(* IEC 61131-3 sources: FDTools/src/Ar/FDTools, 7 files *)

(* ---- DeviceLinker.typ ---- *)
(*
* File: DeviceLinker.typ
* Copyright (c) 2023 Loupe
* https://loupe.team
*
* This file is part of FDTools, licensed under the MIT License.
*
*)

TYPE
	USB_typ : 	STRUCT
		IN : USB_IN_typ;
		OUT : USB_OUT_typ;
		Internal : USB_Internal_typ;
	END_STRUCT;
	USB_IN_typ : 	STRUCT
		PAR : USB_PAR_typ;
		CMD : USB_CMD_typ;
	END_STRUCT;
	USB_PAR_typ : 	STRUCT
		filterInterfaceClass : UINT;
		filterInterfaceSubClass : UINT;
	END_STRUCT;
	USB_CMD_typ : 	STRUCT
		Refresh : BOOL;
		AcknowledgeError : BOOL;
	END_STRUCT;
	USB_OUT_typ : 	STRUCT
		STAT : USB_STAT_typ;
		Interface : ARRAY[0..USB_MAI_NODES]OF STRING[80];
		NumInterfaces : USINT;
		MassStorageDevice : ARRAY[0..USB_MAI_NODES]OF STRING[80];
		NumMassStorages : USINT;
	END_STRUCT;
	USB_STAT_typ : 	STRUCT
		Done : BOOL;
		Busy : BOOL;
		Error : BOOL;
		ErrorID : UINT;
		ErrorString : STRING[80];
	END_STRUCT;
	USB_Internal_typ : 	STRUCT
		State : USB_STATE;
		CMD : USB_CMD_typ;
		STAT : USB_STAT_typ;
		NodeIDList : ARRAY[0..USB_MAI_NODES]OF UDINT;
		NodeList : ARRAY[0..USB_MAI_NODES]OF usbNode_typ;
		DescriptorList : ARRAY[0..USB_MAI_NODES]OF usbDeviceDescr_typ;
		FUB : USB_Internal_FUB_typ;
		NodeIndex : INT;
		AuxInterfaces : ARRAY[0..USB_MAI_NODES]OF STRING[80];
		NumAuxInterface : USINT;
		MassStorageDevices : ARRAY[0..USB_MAI_NODES]OF STRING[80];
		NumMassStorage : USINT;
		RefreshTimer : TON;
	END_STRUCT;
	USB_Internal_FUB_typ : 	STRUCT
		NodeListGet : UsbNodeListGet;
		NodeGet : UsbNodeGet;
		DescriptorGet : UsbDescriptorGet;
	END_STRUCT;
	USB_Selector_Internal_typ : 	STRUCT
		DeviceString : STRING[80];
		iSelectedDevice : STRING[LIST_BOX_STRING_SIZE];
		FileDeviceManager : FileDeviceMgr;
		USBIndex : DINT;
		USBIndexString : STRING[80];
	END_STRUCT;
	FileDeviceMgr_Internal_typ : 	STRUCT
		DevLinkFub : DevLink;
		DevUnlinkFub : DevUnlink;
		iExecute : BOOL;
	END_STRUCT;
	USB_STATE :
		(
		USB_ST_IDLE,
		USB_ST_NODES_GET,
		USB_ST_NODES_READ,
		USB_ST_DESCRIPTORS_READ,
		USB_ST_ERROR,
		USB_ST_
		);
END_TYPE

(* ---- Types.typ ---- *)
(*
* File: Types.typ
* Copyright (c) 2023 Loupe
* https://loupe.team
*
* This file is part of FDTools, licensed under the MIT License.
*
*)

TYPE

END_TYPE

(* ---- USBList.st ---- *)
(*
* File: USBList.st
* Copyright (c) 2023 Loupe
* https://loupe.team
*
* This file is part of FDTools, licensed under the MIT License.
*
*)

(* List all USB nodes *)
FUNCTION USBList

	IF NOT USB.IN.CMD.Refresh AND USB.Internal.CMD.Refresh OR USB.IN.CMD.AcknowledgeError THEN

		USB.IN.CMD.AcknowledgeError:=	0;

		USB.Internal.CMD.Refresh:=0;

		//Reset status
		USB.Internal.STAT.Done:=		0;
		USB.Internal.STAT.Error:=		0;
		USB.Internal.STAT.ErrorID:=		0;
		USB.Internal.STAT.ErrorString:=	'';

	END_IF

	CASE USB.Internal.State OF

		USB_ST_IDLE:

			USB.Internal.STAT.Busy:=		0;

			IF USB.IN.CMD.Refresh AND NOT USB.Internal.CMD.Refresh THEN

				USB.Internal.CMD.Refresh:= 1;

				USB.Internal.State:=	USB_ST_NODES_GET;

				//Reset statuses
				USB.Internal.STAT.Busy:=	1;
				USB.Internal.STAT.Done:=	0;

				//Reset outputs
				USB.Internal.NumMassStorage:=	0;
				USB.Internal.NumAuxInterface:=	0;
				brsmemset(ADR(USB.Internal.MassStorageDevices),0,SIZEOF(USB.Internal.MassStorageDevices));
				brsmemset(ADR(USB.Internal.AuxInterfaces),0,SIZEOF(USB.Internal.AuxInterfaces));

				//Clear out old node data
				brsmemset(ADR(USB.Internal.NodeList),0,SIZEOF(USB.Internal.NodeList));
				brsmemset(ADR(USB.Internal.DescriptorList),0,SIZEOF(USB.Internal.DescriptorList));

			END_IF

		USB_ST_NODES_GET:

			USB.Internal.FUB.NodeListGet.enable:=					1;

			CASE USB.Internal.FUB.NodeListGet.status OF

				ERR_OK:

					USB.Internal.State:=	USB_ST_NODES_READ;

				asusbERR_USB_NOTFOUND:

					USB.Internal.State:=	USB_ST_IDLE;
					USB.Internal.STAT.Done:=	1;

					brsmemcpy(ADR(USB.OUT.Interface),ADR(USB.Internal.AuxInterfaces),SIZEOF(USB.OUT.Interface));
					brsmemcpy(ADR(USB.OUT.MassStorageDevice),ADR(USB.Internal.MassStorageDevices),SIZEOF(USB.OUT.MassStorageDevice));

				ERR_FUB_ENABLE_FALSE,
				ERR_FUB_BUSY:

				ELSE

					USB.Internal.STAT.Error:=		1;
					USB.Internal.STAT.ErrorID:=		USB.Internal.FUB.NodeListGet.status;
					USB.Internal.STAT.ErrorString:=	'Error getting node list';
					USB.Internal.State:=			USB_ST_ERROR;

			END_CASE

		USB_ST_NODES_READ:

			CASE USB.Internal.FUB.NodeGet.status OF

				ERR_OK:

					IF USB.Internal.NodeList[USB.Internal.NodeIndex].interfaceClass = 8 THEN
						USB.Internal.MassStorageDevices[USB.Internal.NumMassStorage]:=	USB.Internal.NodeList[USB.Internal.NodeIndex].ifName;
						USB.Internal.NumMassStorage:=	USB.Internal.NumMassStorage+1;
					ELSIF USB.Internal.NodeList[USB.Internal.NodeIndex].interfaceClass = 255 THEN
						USB.Internal.AuxInterfaces[USB.Internal.NumAuxInterface]:=	USB.Internal.NodeList[USB.Internal.NodeIndex].ifName;
						USB.Internal.NumAuxInterface:=	USB.Internal.NumAuxInterface+1;
					END_IF

					USB.Internal.NodeIndex:=USB.Internal.NodeIndex+1;

					IF USB.Internal.FUB.NodeListGet.listNodes > 0
						AND USB.Internal.FUB.NodeListGet.listNodes > USB.Internal.NodeIndex
						AND USB.Internal.NodeIndex < SIZEOF(USB.Internal.NodeIDList)/SIZEOF(USB.Internal.NodeIDList[0]) THEN

						USB.Internal.FUB.NodeGet.enable:=		1;

					ELSE

						USB.Internal.State:=	USB_ST_DESCRIPTORS_READ;

					END_IF

				ERR_FUB_BUSY:

					//WAIT
					USB.Internal.FUB.NodeGet.enable:=		1;

				ERR_FUB_ENABLE_FALSE:

					USB.Internal.NodeIndex:= 0;
					USB.Internal.FUB.NodeGet.enable:=		1;

				ELSE

					USB.Internal.STAT.Error:=		1;
					USB.Internal.STAT.ErrorID:=		USB.Internal.FUB.NodeGet.status;
					USB.Internal.STAT.ErrorString:=	'Error reading nodes';
					USB.Internal.State:=			USB_ST_ERROR;

			END_CASE

		USB_ST_DESCRIPTORS_READ:

			CASE USB.Internal.FUB.DescriptorGet.status OF
				ERR_OK:

					USB.Internal.NodeIndex:=USB.Internal.NodeIndex+1;

					IF USB.Internal.FUB.NodeListGet.listNodes > 0
						AND USB.Internal.FUB.NodeListGet.listNodes > USB.Internal.NodeIndex
						AND USB.Internal.NodeIndex < SIZEOF(USB.Internal.NodeIDList)/SIZEOF(USB.Internal.NodeIDList[0]) THEN

						USB.Internal.FUB.DescriptorGet.enable:=		1;

					ELSE

						USB.Internal.State:=		USB_ST_IDLE;
						USB.Internal.STAT.Done:=	1;

						brsmemcpy(ADR(USB.OUT.Interface),ADR(USB.Internal.AuxInterfaces),SIZEOF(USB.OUT.Interface));
						brsmemcpy(ADR(USB.OUT.MassStorageDevice),ADR(USB.Internal.MassStorageDevices),SIZEOF(USB.OUT.MassStorageDevice));

						USB.OUT.NumInterfaces:= USB.Internal.NumAuxInterface;
						USB.OUT.NumMassStorages:= USB.Internal.NumMassStorage;

					END_IF

				ERR_FUB_BUSY:

					//WAIT
					USB.Internal.FUB.DescriptorGet.enable:=		1;

				ERR_FUB_ENABLE_FALSE:

					USB.Internal.NodeIndex:= 0;
					USB.Internal.FUB.DescriptorGet.enable:=		1;

				ELSE

					USB.Internal.STAT.Error:=		1;
					USB.Internal.STAT.ErrorID:=		USB.Internal.FUB.DescriptorGet.status;
					USB.Internal.STAT.ErrorString:=	'Error reading node descriptions';
					USB.Internal.State:=			USB_ST_ERROR;

			END_CASE

		USB_ST_ERROR:

			USB.Internal.State:=			USB_ST_IDLE;

	END_CASE

	USB.Internal.RefreshTimer.IN:=	USB.Internal.STAT.Done;
	USB.Internal.RefreshTimer.PT:=	T#3s;
	USB.Internal.RefreshTimer();
	IF USB.Internal.RefreshTimer.Q THEN
		USB.Internal.CMD.Refresh:=	0;
	END_IF

	USB.Internal.FUB.NodeListGet.pBuffer:= 					ADR(USB.Internal.NodeIDList[0]);
	USB.Internal.FUB.NodeListGet.bufferSize:= 				SIZEOF(USB.Internal.NodeIDList);
	USB.Internal.FUB.NodeListGet.filterInterfaceClass:= 	USB.IN.PAR.filterInterfaceClass;
	USB.Internal.FUB.NodeListGet.filterInterfaceSubClass:= 	USB.IN.PAR.filterInterfaceSubClass;
	USB.Internal.FUB.NodeListGet();
	USB.Internal.FUB.NodeListGet.enable:=	0;

	USB.Internal.FUB.NodeGet.nodeId:= 		USB.Internal.NodeIDList[USB.Internal.NodeIndex];
	USB.Internal.FUB.NodeGet.pBuffer:= 		ADR(USB.Internal.NodeList[USB.Internal.NodeIndex]);
	USB.Internal.FUB.NodeGet.bufferSize:= 	SIZEOF(USB.Internal.NodeList[0]);
	USB.Internal.FUB.NodeGet();
	USB.Internal.FUB.NodeGet.enable:=	0;

	USB.Internal.FUB.DescriptorGet.nodeId:= 		USB.Internal.NodeIDList[USB.Internal.NodeIndex];
	USB.Internal.FUB.DescriptorGet.pBuffer:= 		ADR(USB.Internal.DescriptorList[USB.Internal.NodeIndex]);
	USB.Internal.FUB.DescriptorGet.bufferSize:= 	SIZEOF(USB.Internal.DescriptorList[0]);
	//	USB.Internal.FUB.DescriptorGet.descriptorIndex
	//	USB.Internal.FUB.DescriptorGet.descriptorType
	//	USB.Internal.FUB.DescriptorGet.languageId
	//	USB.Internal.FUB.DescriptorGet.requestType
	USB.Internal.FUB.DescriptorGet.descriptorType:= 2;
	USB.Internal.FUB.DescriptorGet();
	USB.Internal.FUB.DescriptorGet.enable:=	0;

	USB.OUT.STAT:=	USB.Internal.STAT;

	USBList:=	USB.OUT.STAT.Done;

END_FUNCTION

(* ---- FDTools.fun ---- *)
(*
* File: FDTools.fun
* Copyright (c) 2023 Loupe
* https://loupe.team
*
* This file is part of FDTools, licensed under the MIT License.
*
*)

FUNCTION USBList : BOOL (*List all USB nodes*) (*$GROUP=User,$GROUPICON=usbms01.front.png*)
	VAR_INPUT
		USB : USB_typ;
	END_VAR
END_FUNCTION

FUNCTION_BLOCK FileDeviceSelector (*Allows the user to select between multiple sources for a file device*) (*$GROUP=User*)
	VAR_INPUT
		Enable : BOOL; (*Enable this function block*)
		FileDevice : STRING[80]; (*File device to link the selected hardware to*)
		pConfiguredDevice : UDINT; (*OPTIONAL: Connect to remnant string variable to reconnect on startup*)
		pUSBList : REFERENCE TO USB_typ; (*OPTIONAL: ADR to USB_typ to populate the list with USB devices*)
		pDirectory : REFERENCE TO STRING[80]; (*OPTIONAL: ADR of String containing the directory to connect to on the CF card*)
		pNetworkConfiguration : REFERENCE TO STRING[80]; (*OPTIONAL: ADR of String containing the network configuration to connect to*)
		Selector : ListBoxFub; (*HMI Connections. Connect this structure to HMI elements to display the results and allow users to select devices.*)
	END_VAR
	VAR_OUTPUT
		Locations : ARRAY[0..12] OF STRING[LIST_BOX_STRING_SIZE]; (*HMI Connections. Connect this array to Listbox or Dropdown to display the results and allow the user to select a device.*)
		status : UINT; (*Status of internal functions*)
		handle : UDINT; (*Handle to unlink in exit routine*)
	END_VAR
	VAR
		internal : USB_Selector_Internal_typ;
		TempString : REFERENCE TO STRING[80];
	END_VAR
END_FUNCTION_BLOCK

FUNCTION_BLOCK FileDeviceMgr (*Links/Unlinks file devices*) (*$GROUP=User*)
	VAR_INPUT
		Execute : BOOL; (*Execute a DevLink*)
		pDevice : UDINT; (*File device to link to hardware*)
		pParam : UDINT; (*Parameter string. See Devlink Help.*)
	END_VAR
	VAR_OUTPUT
		busy : BOOL; (*The function block is working*)
		done : BOOL; (*The function block completed successfully*)
		error : BOOL; (*Error has occured*)
		status : UINT; (*status of devlink/unlink*)
		handle : UDINT; (*Handle to unlink in exit routine*)
	END_VAR
	VAR
		internal : FileDeviceMgr_Internal_typ;
	END_VAR
END_FUNCTION_BLOCK

(* ---- FileDeviceMgr.st ---- *)
(*
* File: FileDeviceMgr.st
* Copyright (c) 2023 Loupe
* https://loupe.team
*
* This file is part of FDTools, licensed under the MIT License.
*
*)

(* Links/Unlinks file devices *)
FUNCTION_BLOCK FileDeviceMgr

	//If execute is false, reset all statuses
	IF NOT Execute THEN

		busy:= 		0;
		done:= 		0;
		status:=	0;
		error:=		0;
		internal.iExecute:=	0;

	END_IF

	//If we have a handle it means that we have devlinked
	//Completion means the user has made a change
	//If so, unlink, then link to the new one
	IF internal.DevUnlinkFub.handle <> 0 AND NOT internal.iExecute AND Execute THEN

		busy:= 		1;
		done:= 		0;
		error:=		0;
		status:= ERR_FUB_BUSY;

		internal.iExecute:=	1;
		internal.DevUnlinkFub.enable:=	1;

	//If we don't have a handle, we can just link.
	//If we actually are linked, it will thow it back to unlink anyway
	ELSIF NOT internal.iExecute AND Execute THEN

		busy:= 		1;
		done:= 		0;
		error:=		0;

		status:= ERR_FUB_BUSY;

		internal.iExecute:=	1;
		internal.DevLinkFub.enable:=		1;

	END_IF

	internal.DevUnlinkFub();

	//When we finish unlinking or have an error, start a link
	IF internal.DevUnlinkFub.status = ERR_OK OR internal.DevUnlinkFub.status = fiERR_SYSTEM THEN
		internal.DevUnlinkFub.enable:=		0;
		internal.DevUnlinkFub.handle:=		0;
		internal.DevLinkFub.enable:=		1;
	ELSIF internal.DevUnlinkFub.status <> ERR_FUB_ENABLE_FALSE THEN
		status:= internal.DevUnlinkFub.status;
		busy:= 		0;
		done:= 		0;
	END_IF

	internal.DevLinkFub.pDevice:=	pDevice;
	internal.DevLinkFub.pParam:=	pParam;
	internal.DevLinkFub();

	CASE internal.DevLinkFub.status OF
		//Link is done, grab the handle for unlinking later
		ERR_OK://Done, grab the handle to unlink later
			internal.DevLinkFub.enable:=		0;
			internal.DevUnlinkFub.handle:= 	internal.DevLinkFub.handle;

			busy:= 		0;
			done:= 		1;

			status:=	internal.DevLinkFub.status;

		//Already linked to different device, unlink and relink when it is finished.
		fiERR_DEVICE_ALREADY_EXIST://Already exist, must unlink first
			//Disable link
			internal.DevLinkFub.enable:=		0;

			//Do an unlink
			IF internal.DevLinkFub.handle <> 0 THEN
				internal.DevUnlinkFub.handle:= internal.DevLinkFub.handle;
				internal.DevUnlinkFub.enable:=	1;
			ELSE
				busy:= 		0;
				done:= 		0;
				status:=	internal.DevLinkFub.status;
			END_IF

		//Working
		ERR_FUB_BUSY:
			status:=	internal.DevLinkFub.status;

		//Do nothing
		ERR_FUB_ENABLE_FALSE:

		fiERR_SYSTEM:
			internal.DevLinkFub.enable:=		0;
			busy:= 		0;
			done:= 		0;
			error:=		1;
			status:=	FileIoGetSysError();

		ELSE

			internal.DevLinkFub.enable:=		0;

			error:=		1;
			busy:= 		0;
			done:= 		0;
			status:=	internal.DevLinkFub.status;
		//OOPS!

	END_CASE

	handle:=	internal.DevUnlinkFub.handle;

END_FUNCTION_BLOCK

(* ---- FileDeviceSelector.st ---- *)
(*
* File: FileDeviceSelector.st
* Copyright (c) 2023 Loupe
* https://loupe.team
*
* This file is part of FDTools, licensed under the MIT License.
*
*)

(* Selects  *)
FUNCTION_BLOCK FileDeviceSelector

	(* Make sure perm memory will link on bootup *)
	(* Check if permanent memory is used, if so assign it *)
	IF Selector.Selection = 0 THEN
		IF pConfiguredDevice <> 0 THEN
			Selector.Selection:=		pConfiguredDevice;
			TempString ACCESS pConfiguredDevice;
			IF TempString <> '' THEN
				internal.FileDeviceManager.Execute:=1;
			END_IF
		ELSE
			Selector.Selection:=		ADR(internal.iSelectedDevice);
		END_IF
	END_IF

	//If a directory location is given, allow the user to select CF
	brsmemset(ADR(Locations),0,SIZEOF(Locations));
	Selector.MaxDP:=0;
	IF ADR(pDirectory) <> 0 THEN
		Locations[Selector.MaxDP]:= 'Disk';
		Selector.MaxDP:=Selector.MaxDP+1;
	END_IF

	//If a network configuration is given, allow the user to select Network share
	IF ADR(pNetworkConfiguration) <> 0 THEN
		Locations[Selector.MaxDP]:= 'Network';
		Selector.MaxDP:=Selector.MaxDP+1;
	END_IF

	//Add any USB storage devices to the list as USBn
	IF ADR(pUSBList) <> 0 THEN
		IF pUSBList.OUT.NumMassStorages > 0 THEN
			FOR internal.USBIndex:=0 TO pUSBList.OUT.NumMassStorages -1 DO
				Locations[Selector.MaxDP]:=	REPLACE(pUSBList.OUT.MassStorageDevice[internal.USBIndex],'USB',3,1);
				Selector.MaxDP:=			Selector.MaxDP+1;
			END_FOR
		END_IF
		//Call selection function block to update screen list
		Selector.Enable:= 	Enable;// AND (pUSBList.OUT.STAT.Done); 	// Only enable while the USB list is done to make sure we don't get flashing, or lose settings between during update
	ELSE
		Selector.Enable:=	Enable;
	END_IF

	Selector.MinDP:=			0;
	Selector.SelectionList:=	ADR(Locations);// Set up the list of device to look at
	Selector();

	IF pConfiguredDevice <> 0 THEN //Check if permanent memory is used, if so copy into internal memory
		brsmemcpy(ADR(internal.iSelectedDevice),pConfiguredDevice,SIZEOF(internal.iSelectedDevice));
	END_IF

	//Completion means the user has made a change
	IF Selector.CompletionDP THEN
		status:=0;
		IF FIND(internal.iSelectedDevice,'USB') <> 0 THEN
			internal.DeviceString:=				CONCAT('/DEVICE=',REPLACE(internal.iSelectedDevice,'/bd',3,1));
			internal.FileDeviceManager.pParam:=	ADR(internal.DeviceString);
			internal.FileDeviceManager.Execute:=1;
		ELSIF FIND(internal.iSelectedDevice,'Disk') <> 0 THEN
			internal.DeviceString:=				CONCAT('/DEVICE=',pDirectory);
			internal.FileDeviceManager.pParam:=	ADR(internal.DeviceString);
			internal.FileDeviceManager.Execute:=1;
		ELSIF FIND(internal.iSelectedDevice,'Network') <> 0 THEN
			internal.FileDeviceManager.pParam:=	ADR(pNetworkConfiguration);
			internal.FileDeviceManager.Execute:=1;
		END_IF
	END_IF

	internal.FileDeviceManager.pDevice:=ADR(FileDevice);
	internal.FileDeviceManager();
	IF internal.FileDeviceManager.error THEN
		status:= internal.FileDeviceManager.status;
	END_IF

	internal.FileDeviceManager.Execute:=	0;

	handle:= internal.FileDeviceManager.handle;

END_FUNCTION_BLOCK

(* ---- Constants.var ---- *)
(*
 * File: Constants.var
 * Copyright (c) 2023 Loupe
 * https://loupe.team
 *
 * This file is part of FDTools, licensed under the MIT License.
 *
  ********************************************************************)

VAR CONSTANT
	USB_MAI_NODES : USINT := 10;
END_VAR
